// Mitsubishi GX Developer project: 11-509_四軸自動供給鎖螺絲機201107181520   PLC: FX1N

PROGRAM MAIN
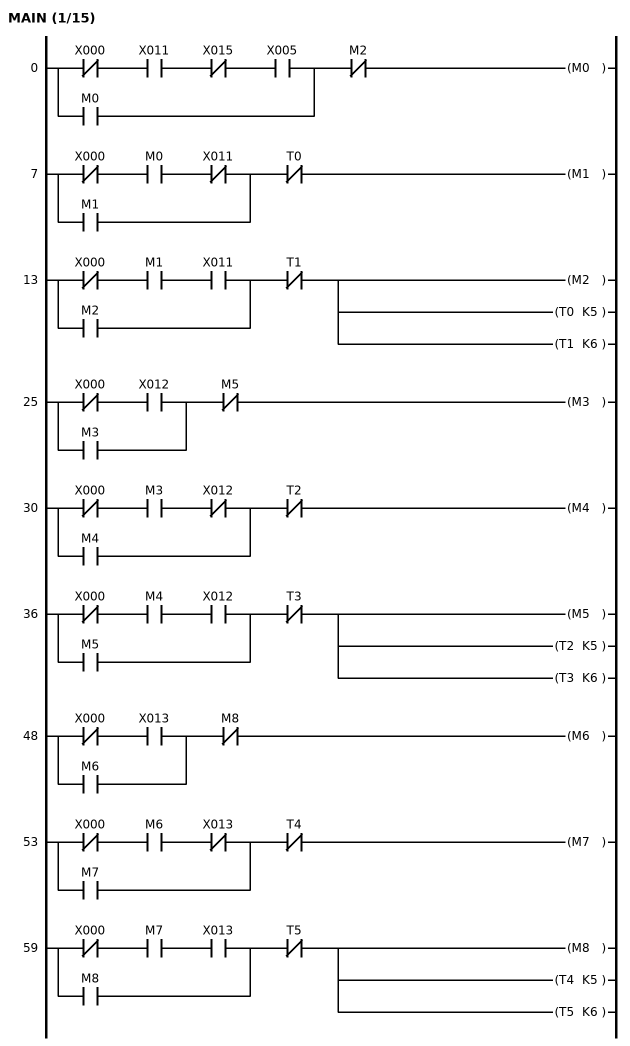
0     LDI     X000
      AND     X011
      ANI     X015
      AND     X005
      OR      M0
      ANI     M2
      OUT     M0
7     LDI     X000
      AND     M0
      ANI     X011
      OR      M1
      ANI     T0
      OUT     M1
13    LDI     X000
      AND     M1
      AND     X011
      OR      M2
      ANI     T1
      OUT     M2
      OUT     T0 K5
      OUT     T1 K6
25    LDI     X000
      AND     X012
      OR      M3
      ANI     M5
      OUT     M3
30    LDI     X000
      AND     M3
      ANI     X012
      OR      M4
      ANI     T2
      OUT     M4
36    LDI     X000
      AND     M4
      AND     X012
      OR      M5
      ANI     T3
      OUT     M5
      OUT     T2 K5
      OUT     T3 K6
48    LDI     X000
      AND     X013
      OR      M6
      ANI     M8
      OUT     M6
53    LDI     X000
      AND     M6
      ANI     X013
      OR      M7
      ANI     T4
      OUT     M7
59    LDI     X000
      AND     M7
      AND     X013
      OR      M8
      ANI     T5
      OUT     M8
      OUT     T4 K5
      OUT     T5 K6
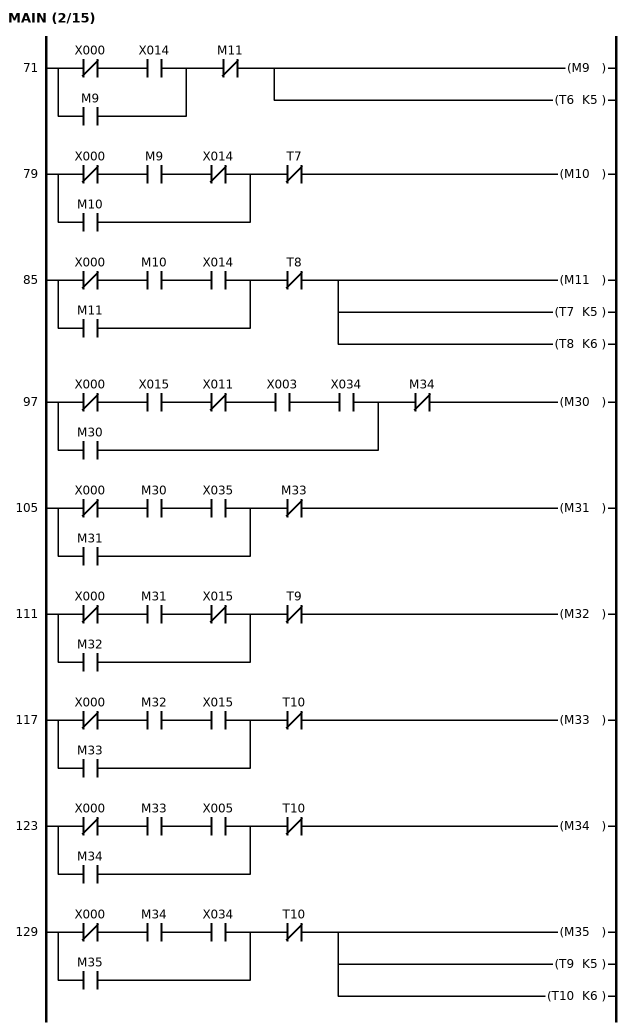
71    LDI     X000
      AND     X014
      OR      M9
      ANI     M11
      OUT     M9
      OUT     T6 K5
79    LDI     X000
      AND     M9
      ANI     X014
      OR      M10
      ANI     T7
      OUT     M10
85    LDI     X000
      AND     M10
      AND     X014
      OR      M11
      ANI     T8
      OUT     M11
      OUT     T7 K5
      OUT     T8 K6
97    LDI     X000
      AND     X015
      ANI     X011
      AND     X003
      AND     X034
      OR      M30
      ANI     M34
      OUT     M30
105   LDI     X000
      AND     M30
      AND     X035
      OR      M31
      ANI     M33
      OUT     M31
111   LDI     X000
      AND     M31
      ANI     X015
      OR      M32
      ANI     T9
      OUT     M32
117   LDI     X000
      AND     M32
      AND     X015
      OR      M33
      ANI     T10
      OUT     M33
123   LDI     X000
      AND     M33
      AND     X005
      OR      M34
      ANI     T10
      OUT     M34
129   LDI     X000
      AND     M34
      AND     X034
      OR      M35
      ANI     T10
      OUT     M35
      OUT     T9 K5
      OUT     T10 K6
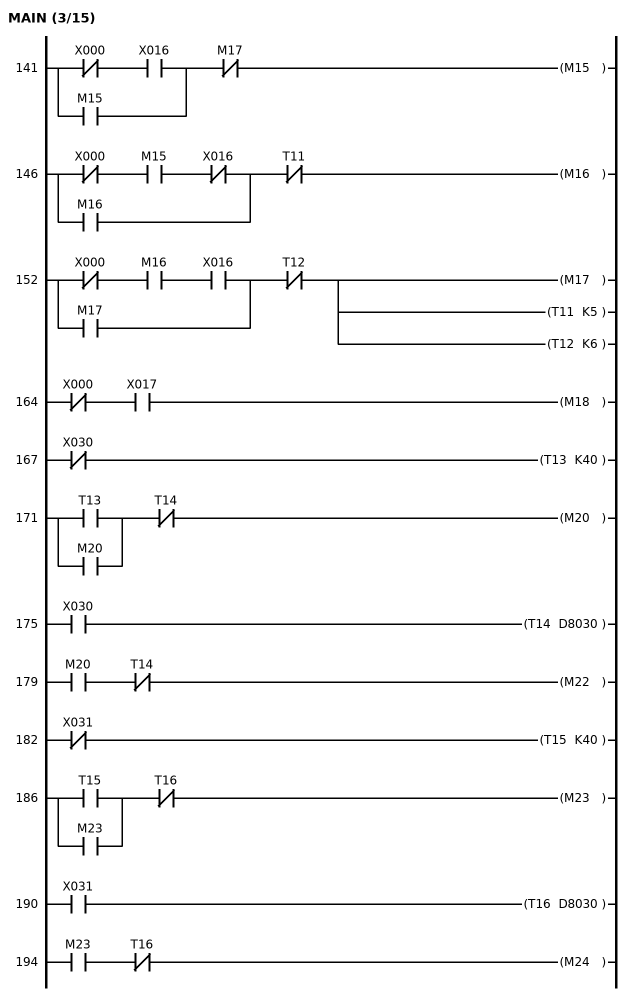
141   LDI     X000
      AND     X016
      OR      M15
      ANI     M17
      OUT     M15
146   LDI     X000
      AND     M15
      ANI     X016
      OR      M16
      ANI     T11
      OUT     M16
152   LDI     X000
      AND     M16
      AND     X016
      OR      M17
      ANI     T12
      OUT     M17
      OUT     T11 K5
      OUT     T12 K6
164   LDI     X000
      AND     X017
      OUT     M18
167   LDI     X030
      OUT     T13 K40
171   LD      T13
      OR      M20
      ANI     T14
      OUT     M20
175   LD      X030
      OUT     T14 D8030
179   LD      M20
      ANI     T14
      OUT     M22
182   LDI     X031
      OUT     T15 K40
186   LD      T15
      OR      M23
      ANI     T16
      OUT     M23
190   LD      X031
      OUT     T16 D8030
194   LD      M23
      ANI     T16
      OUT     M24
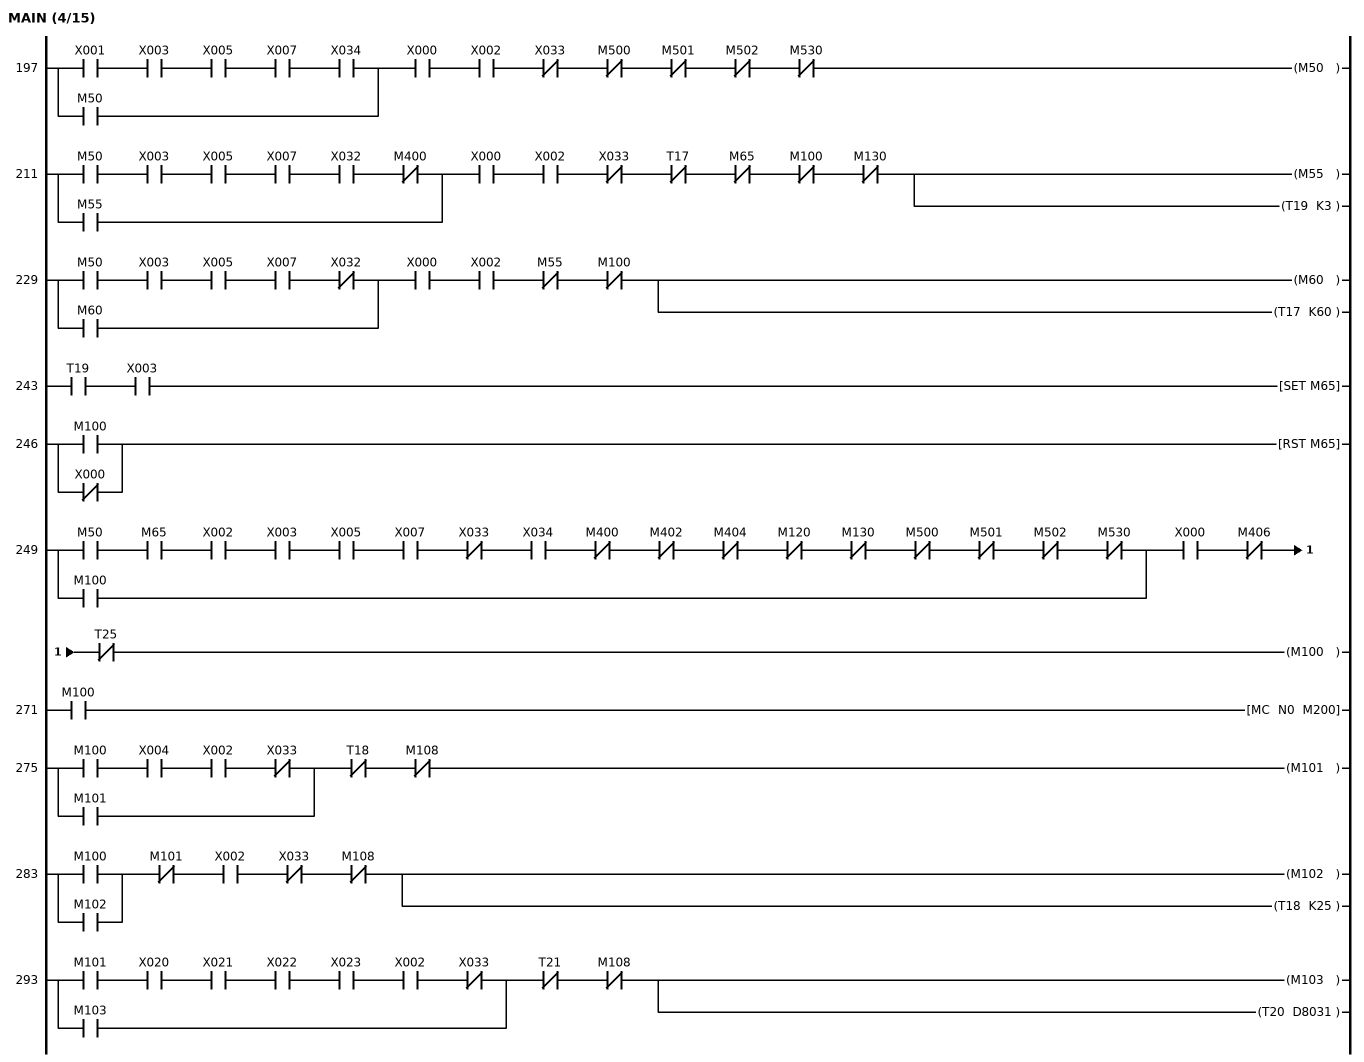
197   LD      X001
      AND     X003
      AND     X005
      AND     X007
      AND     X034
      OR      M50
      AND     X000
      AND     X002
      ANI     X033
      ANI     M500
      ANI     M501
      ANI     M502
      ANI     M530
      OUT     M50
211   LD      M50
      AND     X003
      AND     X005
      AND     X007
      AND     X032
      ANI     M400
      OR      M55
      AND     X000
      AND     X002
      ANI     X033
      ANI     T17
      ANI     M65
      ANI     M100
      ANI     M130
      OUT     M55
      OUT     T19 K3
229   LD      M50
      AND     X003
      AND     X005
      AND     X007
      ANI     X032
      OR      M60
      AND     X000
      AND     X002
      ANI     M55
      ANI     M100
      OUT     M60
      OUT     T17 K60
243   LD      T19
      AND     X003
      SET     M65
246   LD      M100
      ORI     X000
      RST     M65
249   LD      M50
      AND     M65
      AND     X002
      AND     X003
      AND     X005
      AND     X007
      ANI     X033
      AND     X034
      ANI     M400
      ANI     M402
      ANI     M404
      ANI     M120
      ANI     M130
      ANI     M500
      ANI     M501
      ANI     M502
      ANI     M530
      OR      M100
      AND     X000
      ANI     M406
      ANI     T25
      OUT     M100
271   LD      M100
      MC      N0 M200
275   LD      M100
      AND     X004
      AND     X002
      ANI     X033
      OR      M101
      ANI     T18
      ANI     M108
      OUT     M101
283   LD      M100
      OR      M102
      ANI     M101
      AND     X002
      ANI     X033
      ANI     M108
      OUT     M102
      OUT     T18 K25
293   LD      M101
      AND     X020
      AND     X021
      AND     X022
      AND     X023
      AND     X002
      ANI     X033
      OR      M103
      ANI     T21
      ANI     M108
      OUT     M103
      OUT     T20 D8031
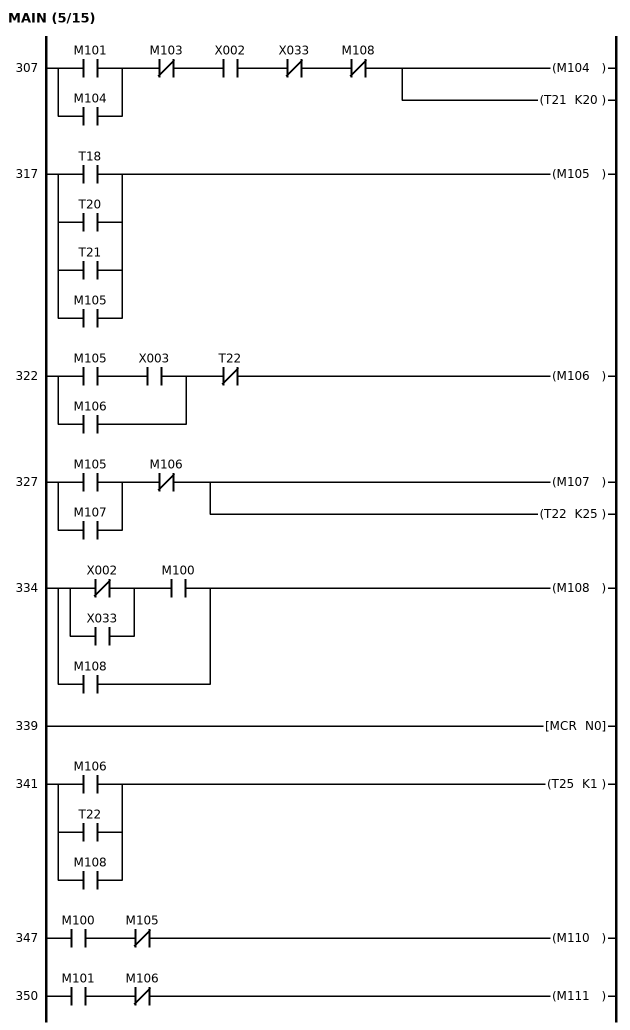
307   LD      M101
      OR      M104
      ANI     M103
      AND     X002
      ANI     X033
      ANI     M108
      OUT     M104
      OUT     T21 K20
317   LD      T18
      OR      T20
      OR      T21
      OR      M105
      OUT     M105
322   LD      M105
      AND     X003
      OR      M106
      ANI     T22
      OUT     M106
327   LD      M105
      OR      M107
      ANI     M106
      OUT     M107
      OUT     T22 K25
334   LDI     X002
      OR      X033
      AND     M100
      OR      M108
      OUT     M108
339   MCR     N0
341   LD      M106
      OR      T22
      OR      M108
      OUT     T25 K1
347   LD      M100
      ANI     M105
      OUT     M110
350   LD      M101
      ANI     M106
      OUT     M111
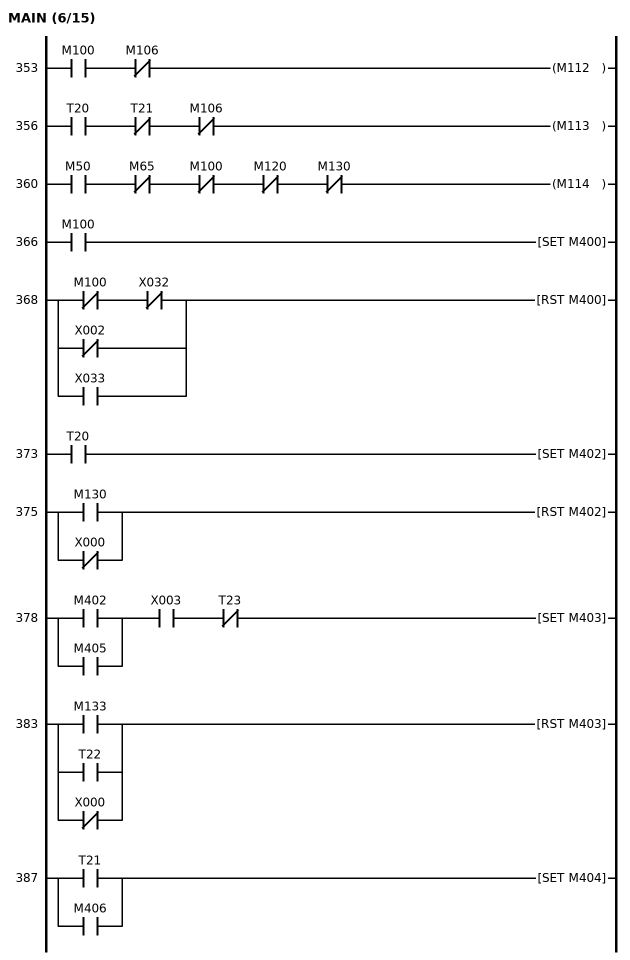
353   LD      M100
      ANI     M106
      OUT     M112
356   LD      T20
      ANI     T21
      ANI     M106
      OUT     M113
360   LD      M50
      ANI     M65
      ANI     M100
      ANI     M120
      ANI     M130
      OUT     M114
366   LD      M100
      SET     M400
368   LDI     M100
      ANI     X032
      ORI     X002
      OR      X033
      RST     M400
373   LD      T20
      SET     M402
375   LD      M130
      ORI     X000
      RST     M402
378   LD      M402
      OR      M405
      AND     X003
      ANI     T23
      SET     M403
383   LD      M133
      OR      T22
      ORI     X000
      RST     M403
387   LD      T21
      OR      M406
      SET     M404
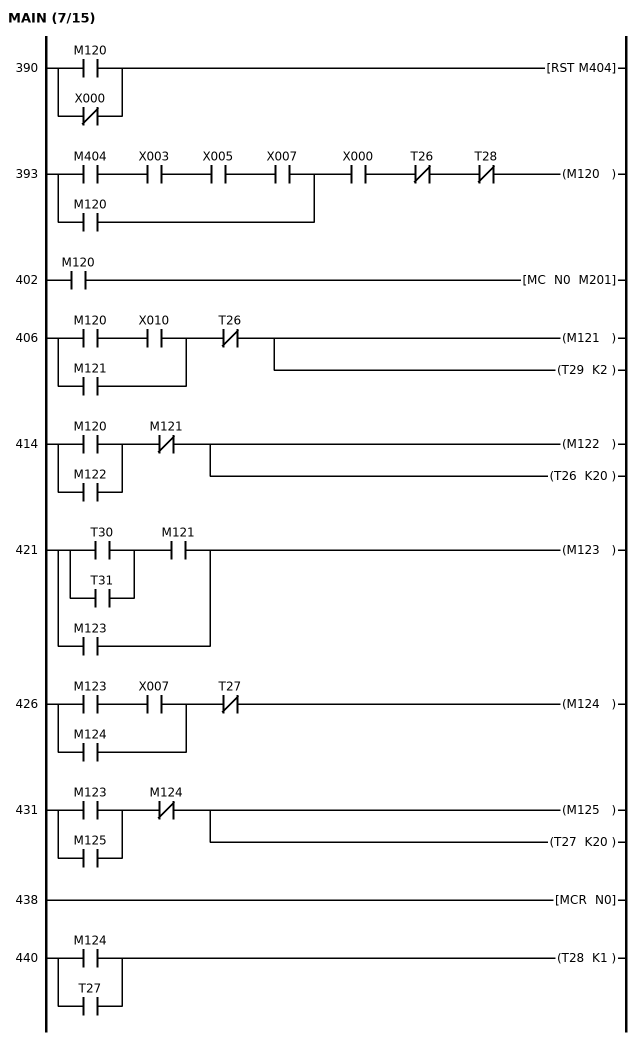
390   LD      M120
      ORI     X000
      RST     M404
393   LD      M404
      AND     X003
      AND     X005
      AND     X007
      OR      M120
      AND     X000
      ANI     T26
      ANI     T28
      OUT     M120
402   LD      M120
      MC      N0 M201
406   LD      M120
      AND     X010
      OR      M121
      ANI     T26
      OUT     M121
      OUT     T29 K2
414   LD      M120
      OR      M122
      ANI     M121
      OUT     M122
      OUT     T26 K20
421   LD      T30
      OR      T31
      AND     M121
      OR      M123
      OUT     M123
426   LD      M123
      AND     X007
      OR      M124
      ANI     T27
      OUT     M124
431   LD      M123
      OR      M125
      ANI     M124
      OUT     M125
      OUT     T27 K20
438   MCR     N0
440   LD      M124
      OR      T27
      OUT     T28 K1
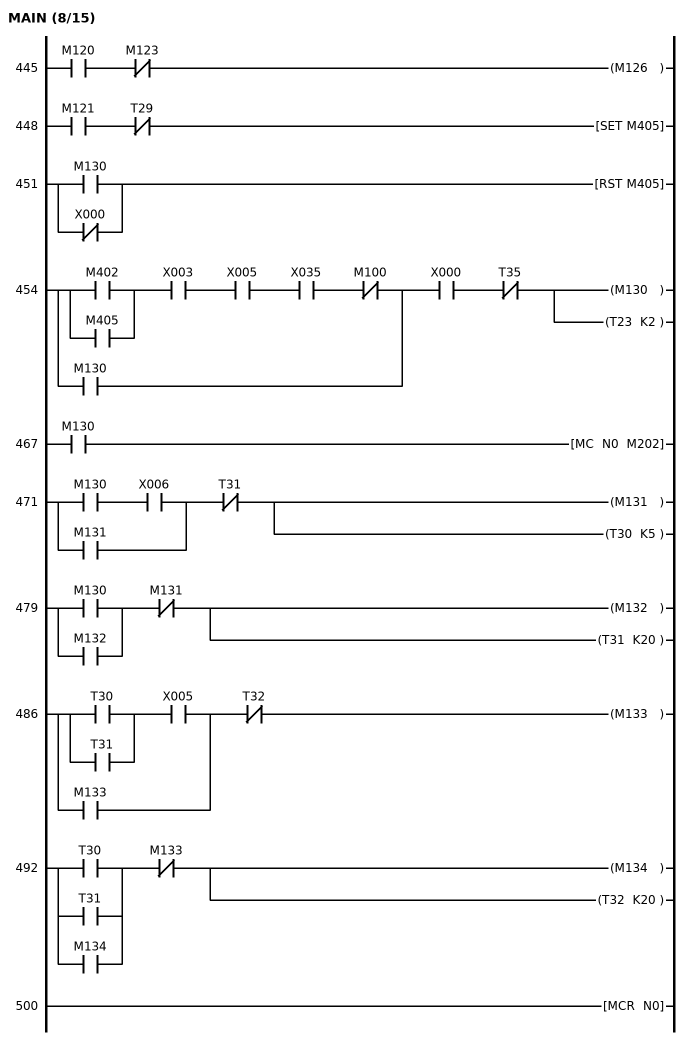
445   LD      M120
      ANI     M123
      OUT     M126
448   LD      M121
      ANI     T29
      SET     M405
451   LD      M130
      ORI     X000
      RST     M405
454   LD      M402
      OR      M405
      AND     X003
      AND     X005
      AND     X035
      ANI     M100
      OR      M130
      AND     X000
      ANI     T35
      OUT     M130
      OUT     T23 K2
467   LD      M130
      MC      N0 M202
471   LD      M130
      AND     X006
      OR      M131
      ANI     T31
      OUT     M131
      OUT     T30 K5
479   LD      M130
      OR      M132
      ANI     M131
      OUT     M132
      OUT     T31 K20
486   LD      T30
      OR      T31
      AND     X005
      OR      M133
      ANI     T32
      OUT     M133
492   LD      T30
      OR      T31
      OR      M134
      ANI     M133
      OUT     M134
      OUT     T32 K20
500   MCR     N0
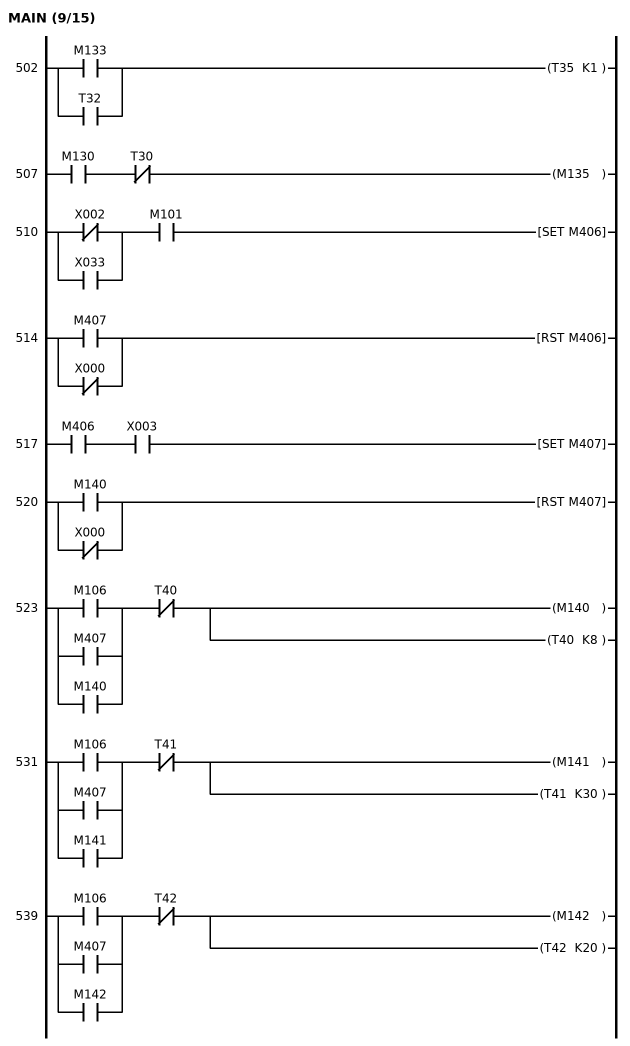
502   LD      M133
      OR      T32
      OUT     T35 K1
507   LD      M130
      ANI     T30
      OUT     M135
510   LDI     X002
      OR      X033
      AND     M101
      SET     M406
514   LD      M407
      ORI     X000
      RST     M406
517   LD      M406
      AND     X003
      SET     M407
520   LD      M140
      ORI     X000
      RST     M407
523   LD      M106
      OR      M407
      OR      M140
      ANI     T40
      OUT     M140
      OUT     T40 K8
531   LD      M106
      OR      M407
      OR      M141
      ANI     T41
      OUT     M141
      OUT     T41 K30
539   LD      M106
      OR      M407
      OR      M142
      ANI     T42
      OUT     M142
      OUT     T42 K20
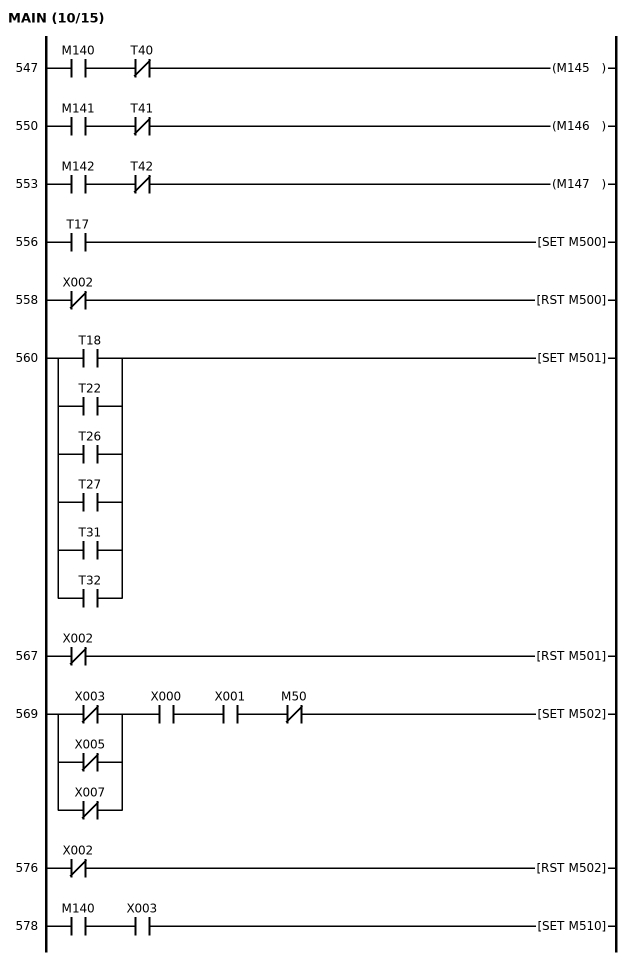
547   LD      M140
      ANI     T40
      OUT     M145
550   LD      M141
      ANI     T41
      OUT     M146
553   LD      M142
      ANI     T42
      OUT     M147
556   LD      T17
      SET     M500
558   LDI     X002
      RST     M500
560   LD      T18
      OR      T22
      OR      T26
      OR      T27
      OR      T31
      OR      T32
      SET     M501
567   LDI     X002
      RST     M501
569   LDI     X003
      ORI     X005
      ORI     X007
      AND     X000
      AND     X001
      ANI     M50
      SET     M502
576   LDI     X002
      RST     M502
578   LD      M140
      AND     X003
      SET     M510
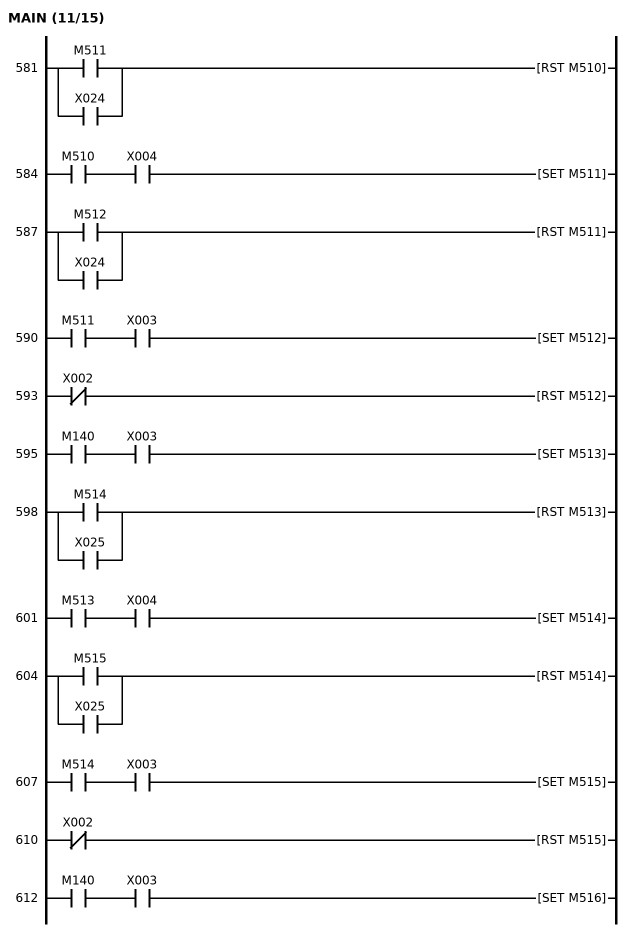
581   LD      M511
      OR      X024
      RST     M510
584   LD      M510
      AND     X004
      SET     M511
587   LD      M512
      OR      X024
      RST     M511
590   LD      M511
      AND     X003
      SET     M512
593   LDI     X002
      RST     M512
595   LD      M140
      AND     X003
      SET     M513
598   LD      M514
      OR      X025
      RST     M513
601   LD      M513
      AND     X004
      SET     M514
604   LD      M515
      OR      X025
      RST     M514
607   LD      M514
      AND     X003
      SET     M515
610   LDI     X002
      RST     M515
612   LD      M140
      AND     X003
      SET     M516
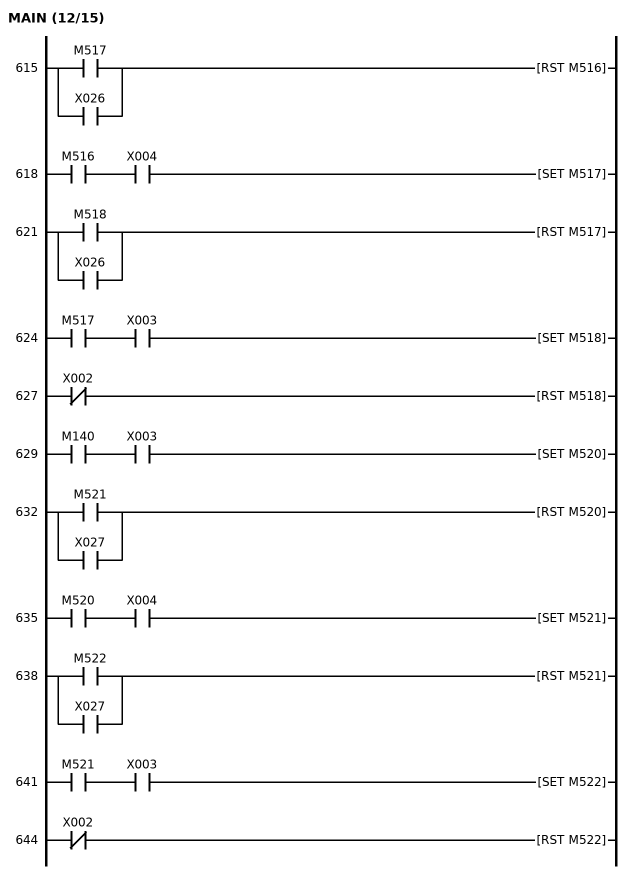
615   LD      M517
      OR      X026
      RST     M516
618   LD      M516
      AND     X004
      SET     M517
621   LD      M518
      OR      X026
      RST     M517
624   LD      M517
      AND     X003
      SET     M518
627   LDI     X002
      RST     M518
629   LD      M140
      AND     X003
      SET     M520
632   LD      M521
      OR      X027
      RST     M520
635   LD      M520
      AND     X004
      SET     M521
638   LD      M522
      OR      X027
      RST     M521
641   LD      M521
      AND     X003
      SET     M522
644   LDI     X002
      RST     M522
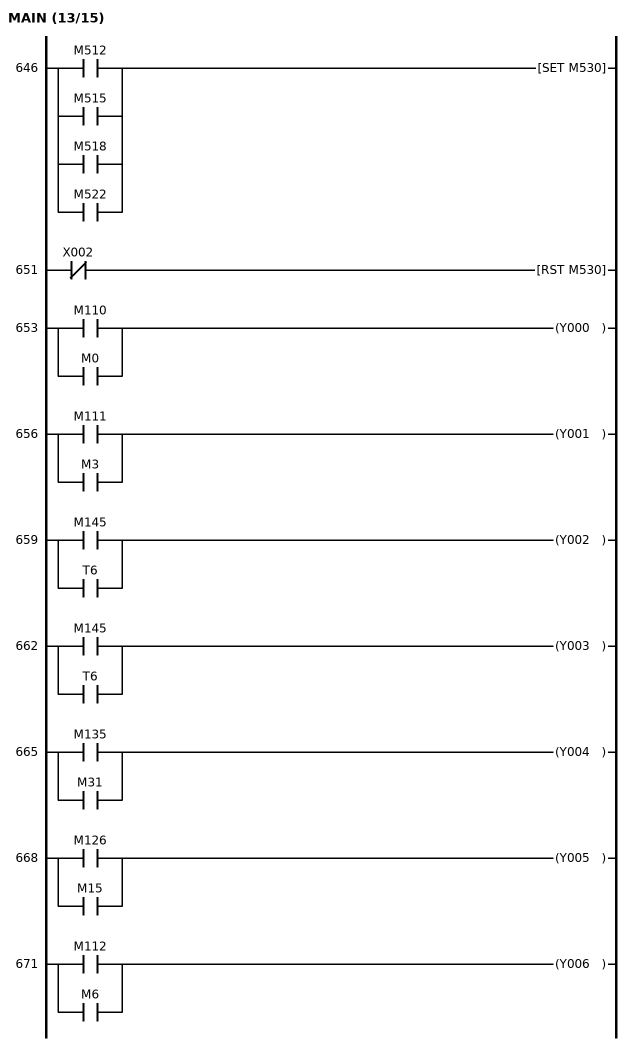
646   LD      M512
      OR      M515
      OR      M518
      OR      M522
      SET     M530
651   LDI     X002
      RST     M530
653   LD      M110
      OR      M0
      OUT     Y000
656   LD      M111
      OR      M3
      OUT     Y001
659   LD      M145
      OR      T6
      OUT     Y002
662   LD      M145
      OR      T6
      OUT     Y003
665   LD      M135
      OR      M31
      OUT     Y004
668   LD      M126
      OR      M15
      OUT     Y005
671   LD      M112
      OR      M6
      OUT     Y006
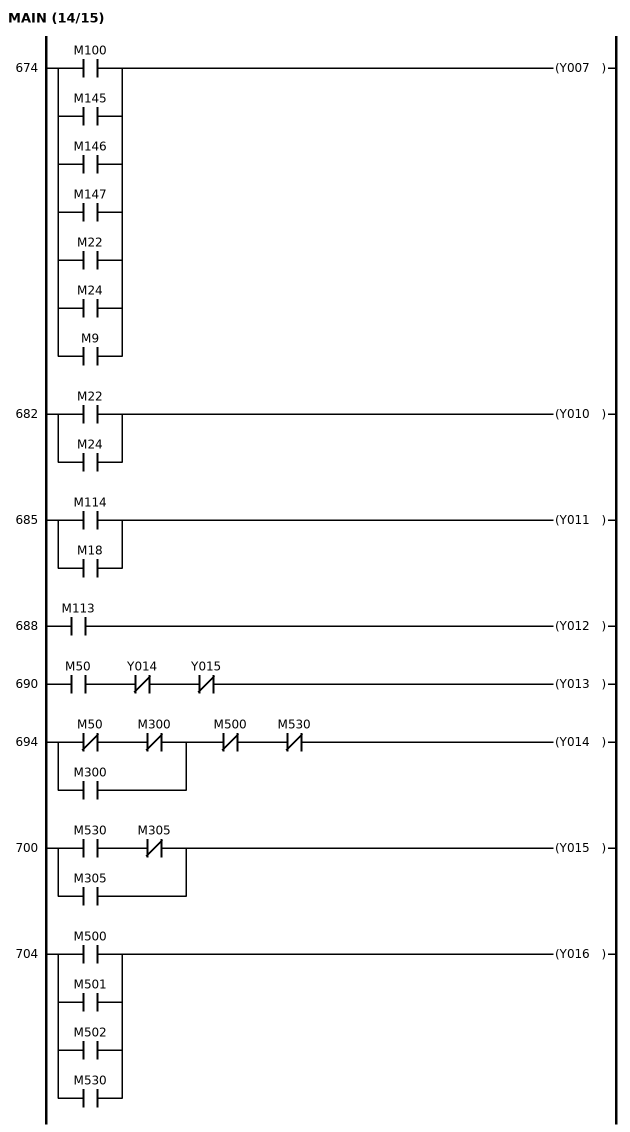
674   LD      M100
      OR      M145
      OR      M146
      OR      M147
      OR      M22
      OR      M24
      OR      M9
      OUT     Y007
682   LD      M22
      OR      M24
      OUT     Y010
685   LD      M114
      OR      M18
      OUT     Y011
688   LD      M113
      OUT     Y012
690   LD      M50
      ANI     Y014
      ANI     Y015
      OUT     Y013
694   LDI     M50
      ANI     M300
      OR      M300
      ANI     M500
      ANI     M530
      OUT     Y014
700   LD      M530
      ANI     M305
      OR      M305
      OUT     Y015
704   LD      M500
      OR      M501
      OR      M502
      OR      M530
      OUT     Y016
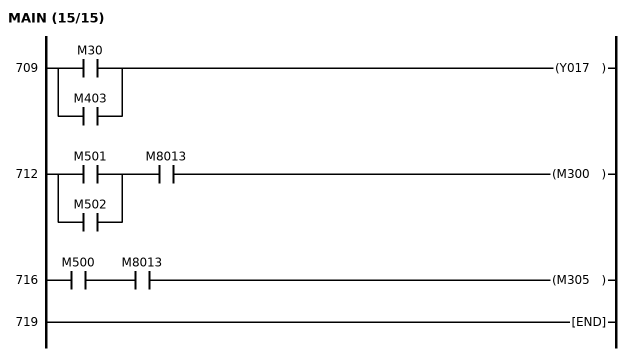
709   LD      M30
      OR      M403
      OUT     Y017
712   LD      M501
      OR      M502
      AND     M8013
      OUT     M300
716   LD      M500
      AND     M8013
      OUT     M305
719   END
END_PROGRAM
